{attribute 'linkalways'} 
{attribute 'no_explicit_call' := 'This FB is a CLASS and must be accessed using methods or properties'}
{attribute 'enable_dynamic_creation'}
FUNCTION_BLOCK BaseElement EXTENDS Disposable IMPLEMENTS I_EventEmitter, I_BaseElement
VAR
	inputPorts : InputPorts;
	outputPorts : OutputPorts;
	parameters : Parameters;
	contents : Contents;
	errors : Errors;
	extensions : Extensions;
	metadata : Metadata;
	eventEmitter : EventEmitter;
	disposables : Stack;
END_VAR

METHOD AddContent
VAR_INPUT
	Content : I_Content;
END_VAR
RegisterContent(Content);
END_METHOD

METHOD AddDataAsContent
VAR_INPUT
	Name : T_MAXSTRING;
	Data : I_Datatype;
END_VAR
VAR
	newContent : I_Content;
END_VAR
newContent := CreateContent(Name, Data);
RegisterDisposableToSelf(newContent);
END_METHOD

METHOD AddDataAsInputPort
VAR_INPUT
	Name : T_MAXSTRING;
	Data : I_Datatype;
END_VAR
VAR
	newInputPort : I_InputPort;
END_VAR
newInputPort := CreateInputPort(Name, Data);
RegisterDisposableToSelf(newInputPort);
END_METHOD

METHOD AddDataAsOutputPort
VAR_INPUT
	Name : T_MAXSTRING;
	Data : I_Datatype;
END_VAR
VAR
	newOutputPort : I_OutputPort;
END_VAR
newOutputPort := CreateOutputPort(Name, Data);
RegisterDisposableToSelf(newOutputPort);
END_METHOD

METHOD AddDataAsParameter
VAR_INPUT
	Name : T_MAXSTRING;
	Data : I_Datatype;
END_VAR
VAR
	newParameter : I_Parameter;
END_VAR
newParameter := CreateParameter(Name, Data);
RegisterDisposableToSelf(newParameter);
END_METHOD

METHOD AddError
VAR_INPUT
	Error : I_Error;
END_VAR
RegisterError(Error);
END_METHOD

METHOD AddExtension
VAR_INPUT
	Extension : I_Extension;
END_VAR
RegisterExtension(Extension);
END_METHOD

METHOD AddInputPort
VAR_INPUT
	InputPort : I_InputPort;
END_VAR
RegisterInputPort(InputPort);
END_METHOD

METHOD AddMetadatum
VAR_INPUT
	Metadatum : I_Metadatum;
END_VAR
RegisterMetadatum(Metadatum);
END_METHOD

METHOD AddOutputPort
VAR_INPUT
	OutputPort : I_OutputPort;
END_VAR
RegisterOutputPort(OutputPort);
END_METHOD

METHOD AddParameter
VAR_INPUT
	Parameter : I_Parameter;
END_VAR
RegisterParameter(Parameter);
END_METHOD

METHOD PROTECTED CreateContent : I_Content
VAR_INPUT
	ContentName : T_MAXSTRING;
	ContentData : I_Datatype;
END_VAR
VAR
	pContent : POINTER TO Content;
END_VAR
pContent := __NEW(Content(Name := ContentName, Data := ContentData, Parent := THIS^));
CreateContent := pContent^;
END_METHOD

METHOD PROTECTED CreateInputPort : I_InputPort
VAR_INPUT
	InputPortName : T_MAXSTRING;
	InputPortData : I_Datatype;
END_VAR
VAR
	pInputPort: POINTER TO InputPort;
END_VAR
pInputPort := __NEW(InputPort(Name := InputPortName, Data := InputPortData, Parent := THIS^));
CreateInputPort := pInputPort^;
END_METHOD

METHOD PROTECTED CreateOutputPort : I_OutputPort
VAR_INPUT
	OutputPortName : T_MAXSTRING;
	OutputPortData : I_Datatype;
END_VAR
VAR
	pOutputPort : POINTER TO OutputPort;
END_VAR
pOutputPort := __NEW(OutputPort(Name := OutputPortName, Data := OutputPortData, Parent := THIS^));
CreateOutputPort := pOutputPort^;
END_METHOD

METHOD PROTECTED CreateParameter : I_Parameter
VAR_INPUT
	ParameterName : T_MAXSTRING;
	ParameterData : I_Datatype;
END_VAR
VAR
	pParameter : POINTER TO Parameter;
END_VAR
pParameter := __NEW(Parameter(Name := ParameterName, Data := ParameterData, Parent := THIS^));
CreateParameter := pParameter^;
END_METHOD

METHOD PROTECTED DisposeAll : BOOL
VAR_INPUT
END_VAR
VAR
	disposable : I_Disposable;
END_VAR
WHILE disposables.TryPop(disposable) DO
	disposable.Dispose();
END_WHILE
END_METHOD

METHOD PROTECTED EmitOnContentAddedEvent
VAR_INPUT
	Content : I_Content;
END_VAR
VAR
	pContentAddedEvent : POINTER TO ContentAddedEvent;
END_VAR
IF Content = 0 THEN
	RETURN;
END_IF

pContentAddedEvent := __NEW(ContentAddedEvent(TargetContent := Content));
eventEmitter.Emit('OnContentAdded',pContentAddedEvent^);
pContentAddedEvent^.Dispose();
END_METHOD

METHOD PROTECTED EmitOnErrorAddedEvent
VAR_INPUT
	Error : I_Error;
END_VAR
VAR
	pErrorAddedEvent : POINTER TO ErrorAddedEvent;
END_VAR
IF Error = 0 THEN
	RETURN;
END_IF

pErrorAddedEvent := __NEW(ErrorAddedEvent(TargetError := Error));
eventEmitter.Emit('OnErrorAdded',pErrorAddedEvent^);
pErrorAddedEvent^.Dispose();
END_METHOD

METHOD PROTECTED EmitOnExtensionAddedEvent
VAR_INPUT
	Extension : I_Extension;
END_VAR
VAR
	pExtensionAddedEvent : POINTER TO ExtensionAddedEvent;
END_VAR
IF Extension = 0 THEN
	RETURN;
END_IF

pExtensionAddedEvent := __NEW(ExtensionAddedEvent(TargetExtension := Extension));
eventEmitter.Emit('OnExtensionAdded',pExtensionAddedEvent^);
pExtensionAddedEvent^.Dispose();
END_METHOD

METHOD PROTECTED EmitOnInputPortAddedEvent
VAR_INPUT
	InputPort : I_InputPort;
END_VAR
VAR
	pInputPortAddedEvent : POINTER TO InputPortAddedEvent;
END_VAR
IF InputPort = 0 THEN
	RETURN;
END_IF

pInputPortAddedEvent := __NEW(InputPortAddedEvent(TargetInputPort := InputPort));
eventEmitter.Emit('OnInputPortAdded',pInputPortAddedEvent^);
pInputPortAddedEvent^.Dispose();
END_METHOD

METHOD PROTECTED EmitOnMetadatumAddedEvent
VAR_INPUT
	Metadatum : I_Metadatum;
END_VAR
VAR
	pMetadatumAddedEvent : POINTER TO MetadatumAddedEvent;
END_VAR
IF Metadatum = 0 THEN
	RETURN;
END_IF

pMetadatumAddedEvent := __NEW(MetadatumAddedEvent(TargetMetadatum := Metadatum));
eventEmitter.Emit('OnMetadatumAdded',pMetadatumAddedEvent^);
pMetadatumAddedEvent^.Dispose();
END_METHOD

METHOD PROTECTED EmitOnOutputPortAddedEvent
VAR_INPUT
	OutputPort : I_OutputPort;
END_VAR
VAR
	pOutputPortAddedEvent : POINTER TO OutputPortAddedEvent;
END_VAR
IF OutputPort = 0 THEN
	RETURN;
END_IF

pOutputPortAddedEvent := __NEW(OutputPortAddedEvent(TargetOutputPort := OutputPort));
eventEmitter.Emit('OnOutputPortAdded',pOutputPortAddedEvent^);
pOutputPortAddedEvent^.Dispose();
END_METHOD

METHOD PROTECTED EmitOnParameterAddedEvent
VAR_INPUT
	Parameter : I_Parameter;
END_VAR
VAR
	pParameterAddedEvent : POINTER TO PropertyAddedEvent;
END_VAR
IF Parameter = 0 THEN
	RETURN;
END_IF

pParameterAddedEvent := __NEW(PropertyAddedEvent(TargetProperty := Parameter));
eventEmitter.Emit('OnParameterAdded',pParameterAddedEvent^);
pParameterAddedEvent^.Dispose();
END_METHOD

METHOD FB_exit : BOOL
VAR_INPUT
	bInCopyCode : BOOL; // if TRUE, the exit method is called for exiting an instance that is copied afterwards (online change).
END_VAR
IF bInCopyCode THEN
	RETURN;
END_IF

DisposeAll();
END_METHOD

METHOD PUBLIC GetContents : I_Contents
VAR_INPUT
END_VAR
GetContents := contents;
END_METHOD

METHOD PUBLIC GetErrors : I_Errors
VAR_INPUT
END_VAR
GetErrors := errors;
END_METHOD

METHOD PUBLIC GetExtensions : I_Extensions
VAR_INPUT
END_VAR
GetExtensions := extensions;
END_METHOD

METHOD PUBLIC GetInputPorts : I_InputPorts
VAR_INPUT
END_VAR
GetInputPorts := inputPorts;
END_METHOD

METHOD PUBLIC GetMetadata : I_Metadata
VAR_INPUT
END_VAR
GetMetadata := metadata;
END_METHOD

METHOD PUBLIC GetOutputPorts : I_OutputPorts
VAR_INPUT
END_VAR
GetOutputPorts := outputPorts;
END_METHOD

METHOD PUBLIC GetParameters : I_Parameters
VAR_INPUT
END_VAR
GetParameters := parameters;
END_METHOD

METHOD PUBLIC OffEvent
VAR_INPUT
	EventName : T_MaxString;
	EventHandler : I_EventHandler;
END_VAR
eventEmitter.OffEvent(EventName, EventHandler);
END_METHOD

METHOD PUBLIC OnceEvent
VAR_INPUT
	EventName : T_MaxString;
	EventHandler : I_EventHandler;
END_VAR
eventEmitter.OnceEvent(EventName, EventHandler);
END_METHOD

METHOD PUBLIC OnEvent
VAR_INPUT
	EventName : T_MaxString;
	EventHandler : I_EventHandler;
END_VAR
eventEmitter.OnEvent(EventName, EventHandler);
END_METHOD

METHOD PROTECTED RegisterContent
VAR_INPUT
	Content : I_Content;
END_VAR
contents.Insert(Content);
EmitOnContentAddedEvent(Content);
END_METHOD

METHOD PROTECTED RegisterDisposableToSelf
VAR_INPUT
	Disposable : I_Disposable;
END_VAR
disposables.Push(Disposable);
END_METHOD

METHOD PROTECTED RegisterError
VAR_INPUT
	Error : I_Error;
END_VAR
errors.Insert(Error);
EmitOnErrorAddedEvent(Error);
END_METHOD

METHOD PROTECTED RegisterExtension
VAR_INPUT
	Extension : I_Extension;
END_VAR
extensions.Insert(Extension);
EmitOnExtensionAddedEvent(Extension);
END_METHOD

METHOD PROTECTED RegisterInputPort
VAR_INPUT
	InputPort : I_InputPort;
END_VAR
inputPorts.Insert(InputPort);
EmitOnInputPortAddedEvent(InputPort);
END_METHOD

METHOD PROTECTED RegisterMetadatum
VAR_INPUT
	Metadatum : I_Metadatum;
END_VAR
metadata.Insert(Metadatum);
EmitOnMetadatumAddedEvent(Metadatum);
END_METHOD

METHOD PROTECTED RegisterOutputPort
VAR_INPUT
	OutputPort : I_OutputPort;
END_VAR
outputPorts.Insert(OutputPort);
EmitOnOutputPortAddedEvent(OutputPort);
END_METHOD

METHOD PROTECTED RegisterParameter
VAR_INPUT
	Parameter : I_Parameter;
END_VAR
parameters.Insert(Parameter);
EmitOnParameterAddedEvent(Parameter);
END_METHOD

METHOD PUBLIC SerializeWith
VAR_INPUT
	Serializer : I_Serializer;
END_VAR
Serializer.StartObject();
Serializer.AddKeyObject('inputPorts',inputPorts);
Serializer.AddKeyObject('outputPorts',outputPorts);
Serializer.AddKeyObject('parameters',parameters);
Serializer.AddKeyObject('contents',contents);
Serializer.AddKeyObject('errors',errors);
Serializer.AddKeyObject('extensions',extensions);
Serializer.AddKeyObject('metadata',metadata);
Serializer.EndObject();
END_METHOD

METHOD PROTECTED TryDeserializeExtensionsFrom : BOOL
VAR_INPUT
	Deserializer : I_Deserializer;
END_VAR
VAR
	extensionsDeserializer : I_Deserializer;
END_VAR
extensionsDeserializer := Deserializer.GetKey('extensions');
extensions.TryDeserializeFrom(extensionsDeserializer);
END_METHOD

METHOD PUBLIC TryDeserializeFrom : BOOL
VAR_INPUT
	Deserializer : I_Deserializer;
END_VAR
TryDeserializeFrom := 
	TryDeserializeParametersFrom(Deserializer) AND 
	TryDeserializeExtensionsFrom(Deserializer);
END_METHOD

METHOD PROTECTED TryDeserializeParametersFrom : BOOL
VAR_INPUT
	Deserializer : I_Deserializer;
END_VAR
VAR
	parametersDeserializer : I_Deserializer;
END_VAR
parametersDeserializer := Deserializer.GetKey('properties');
parameters.TryDeserializeFrom(parametersDeserializer);
END_METHOD

METHOD PUBLIC TryGetContentByName : BOOL
VAR_INPUT
	Name : T_MAXSTRING;
	Destination : REFERENCE TO I_Content;
END_VAR
VAR
	extensionName : T_MAXSTRING;
	extension : I_Extension;
	contentName : T_MAXSTRING;
END_VAR
IF Not HasExtensionNamespace(Name) THEN
	TryGetContentByName := contents.TryGetByName(Name,Destination);
	RETURN;
END_IF

extensionName := RemoveLastSegmentFromNamespace(Name);
contentName := GetLastSegmentFromNamespace(Name);

IF NOT TryGetExtensionByName(extensionName, extension) THEN
	RETURN;
END_IF

TryGetContentByName := extension.TryGetContentByName(contentName, Destination);
END_METHOD

METHOD PUBLIC TryGetExtensionByName : BOOL
VAR_INPUT
	Name : T_MAXSTRING;
	Destination : REFERENCE TO I_Extension;
END_VAR
VAR
	extensionName : T_MAXSTRING;
	remainingName : T_MAXSTRING;
	extension : I_Extension;
END_VAR
IF Not HasExtensionNamespace(Name) THEN
	TryGetExtensionByName := extensions.TryGetByName(Name, Destination);
	RETURN;
END_IF

extensionName := RemoveLastSegmentFromNamespace(Name);
remainingName := GetLastSegmentFromNamespace(Name);

IF NOT this^.TryGetExtensionByName(extensionName, extension) THEN
	RETURN;
END_IF

TryGetExtensionByName := extension.TryGetExtensionByName(remainingName, Destination);
END_METHOD

METHOD PUBLIC TryGetInputPortByName : BOOL
VAR_INPUT
	Name : T_MAXSTRING;
	Destination : REFERENCE TO I_InputPort;
END_VAR
VAR
	extensionName : T_MAXSTRING;
	extension : I_Extension;
	portName : T_MAXSTRING;
END_VAR
IF NOT HasExtensionNamespace(Name) THEN
	TryGetInputPortByName := inputPorts.TryGetByName(Name,Destination);
	RETURN;
END_IF

extensionName := RemoveLastSegmentFromNamespace(Name);
portName := GetLastSegmentFromNamespace(Name);

IF NOT TryGetExtensionByName(extensionName, extension) THEN
	RETURN;
END_IF

TryGetInputPortByName := extension.TryGetInputPortByName(portName, Destination);
END_METHOD

METHOD PUBLIC TryGetMetadatumByName : BOOL
VAR_INPUT
	Name : T_MAXSTRING;
	Destination : REFERENCE TO I_Metadatum;
END_VAR
VAR
	extensionName : T_MAXSTRING;
	extension : I_Extension;
	metadatumName : T_MAXSTRING;
END_VAR
IF NOT HasExtensionNamespace(Name) THEN
	TryGetMetadatumByName := metadata.TryGetByName(Name,Destination);
	RETURN;
END_IF

extensionName := RemoveLastSegmentFromNamespace(Name);
metadatumName := GetLastSegmentFromNamespace(Name);

IF NOT TryGetExtensionByName(extensionName, extension) THEN
	RETURN;
END_IF

TryGetMetadatumByName := extension.TryGetMetadatumByName(metadatumName, Destination);
END_METHOD

METHOD PUBLIC TryGetOutputPortByName : BOOL
VAR_INPUT
	Name : T_MAXSTRING;
	Destination : REFERENCE TO I_OutputPort;
END_VAR
VAR
	extensionName : T_MAXSTRING;
	extension : I_Extension;
	portName : T_MAXSTRING;
END_VAR
IF NOT HasExtensionNamespace(Name) THEN
	TryGetOutputPortByName := outputPorts.TryGetByName(Name,Destination);
	RETURN;
END_IF

extensionName := RemoveLastSegmentFromNamespace(Name);
portName := GetLastSegmentFromNamespace(Name);

IF NOT TryGetExtensionByName(extensionName, extension) THEN
	RETURN;
END_IF

TryGetOutputPortByName := extension.TryGetOutputPortByName(portName, Destination);
END_METHOD

METHOD PUBLIC TryGetParameterByName : BOOL
VAR_INPUT
	Name : T_MAXSTRING;
	Destination : REFERENCE TO I_Parameter;
END_VAR
VAR
	extensionName : T_MAXSTRING;
	extension : I_Extension;
	parameterName : T_MAXSTRING;
END_VAR
IF Not HasExtensionNamespace(Name) THEN
	TryGetParameterByName := parameters.TryGetByName(Name,Destination);
	RETURN;
END_IF

extensionName := RemoveLastSegmentFromNamespace(Name);
parameterName := GetLastSegmentFromNamespace(Name);

IF NOT TryGetExtensionByName(extensionName, extension) THEN
	RETURN;
END_IF

TryGetParameterByName := extension.TryGetParameterByName(parameterName, Destination);
END_METHOD

END_FUNCTION_BLOCK

(* stored: Version 1.1.0.1, ProductVersion 3.1.4024.12
   POU BaseElement: Id {65854565-5a7d-02f2-2709-1993949f09a2}, SpecialFunc None
   Folder Destructor: Id {8396773a-400b-43fa-8a6d-bbe9b1d6ecd3}
   Folder Protected: Id {48a95438-1d6b-0ead-29c1-c8ed21d5c5f8}
   Method AddContent: Id {65c5bac1-a3d0-002c-2cbe-a7b37fe3b45b}
   Method AddDataAsContent: Id {56e24acc-fc0e-4690-8a55-08bdbfb1feb3}
   Method AddDataAsInputPort: Id {4722f8e7-5165-4f79-9bed-1e281e05abb9}
   Method AddDataAsOutputPort: Id {dca4d70a-2386-4112-8b2e-e77a6edffbe6}
   Method AddDataAsParameter: Id {36004062-8b8a-4b3b-89b0-5b74d6f6bc9b}
   Method AddError: Id {4bbd3a02-551d-0fb6-097a-770c7ef9b02a}
   Method AddExtension: Id {12d5c379-9667-00ca-1a5e-59797e6bc21d}
   Method AddInputPort: Id {8aebf87c-0955-0d8e-0a5d-38af87c0ae0d}
   Method AddMetadatum: Id {371a7ce8-9ce1-0df1-08ad-592aac14c8db}
   Method AddOutputPort: Id {8d1e0294-027c-08af-0add-f26ea3b4e6b4}
   Method AddParameter: Id {22e10c77-042d-014a-1131-e8a94df32d37}
   Method CreateContent: Id {821b80ea-fa86-42dc-87c5-a687613888b2}
   Method CreateInputPort: Id {e170d3ea-2856-48fe-99f4-ab4fbe2d037c}
   Method CreateOutputPort: Id {bf3f2d9c-860a-4f77-a8dc-28e59fb38283}
   Method CreateParameter: Id {1ddc001e-24d0-48f3-b9e0-ff7f17397987}
   Method DisposeAll: Id {cb49ffb4-2cda-42c6-89fb-5c15e2905cfd}
   Method EmitOnContentAddedEvent: Id {982e38f9-d0ec-0d68-23b9-1014864696d7}
   Method EmitOnErrorAddedEvent: Id {5f18b0c5-cc95-02f2-100c-2ef3ad7e1a71}
   Method EmitOnExtensionAddedEvent: Id {f402631d-81f9-0a12-03bc-2a0bfe9edd1d}
   Method EmitOnInputPortAddedEvent: Id {999a27ba-e180-0c81-3fd5-7f26e1dcafa9}
   Method EmitOnMetadatumAddedEvent: Id {5e041b08-cbe4-0f2d-0996-099d35827b7a}
   Method EmitOnOutputPortAddedEvent: Id {0092de63-0b62-04d1-3582-5fcf00057f98}
   Method EmitOnParameterAddedEvent: Id {ef9a119a-00ba-01e3-3336-a5211fd3bf30}
   Method FB_exit: Id {6b932cb7-4150-4273-8597-9e500c0eaf5e}
   Method GetContents: Id {81f125c5-c13a-026a-3de6-aa1ebc6668c9}
   Method GetErrors: Id {0627fae9-4882-0c55-17d9-c59657d05963}
   Method GetExtensions: Id {be4c5a1a-53d3-0499-27b1-32409495df61}
   Method GetInputPorts: Id {7de9fbdd-fa4d-0d6e-0b3b-13feae4c89d5}
   Method GetMetadata: Id {dbde985b-051a-0727-258a-c2925ede1d19}
   Method GetOutputPorts: Id {f627e22a-94e0-005f-10c4-a9f76f86d6e8}
   Method GetParameters: Id {f803076c-9d09-002d-18bd-949f984e4d58}
   Method OffEvent: Id {3826f2c5-8817-085f-32d4-f42ca6017d84}
   Method OnceEvent: Id {c0653d6f-a473-06ad-0f4f-23e16a4ab170}
   Method OnEvent: Id {f1641710-5271-0c90-204a-d8ba0111dbe4}
   Method RegisterContent: Id {b67f9558-618d-4bfd-b717-886a90f2936b}
   Method RegisterDisposableToSelf: Id {818ccf26-b9c1-40b3-8452-6ca75c4281c5}
   Method RegisterError: Id {65cdee1a-3625-45b6-bfd7-f72ce4f3aef5}
   Method RegisterExtension: Id {f527d3d7-1297-4450-90c8-dbf3475e7a3d}
   Method RegisterInputPort: Id {a90f95fc-e99b-45fe-ad6f-5621929e0e45}
   Method RegisterMetadatum: Id {c3fb64d8-e827-436e-9972-728da0497a0c}
   Method RegisterOutputPort: Id {8be6e625-9fd4-44dd-a437-f152d0338e1b}
   Method RegisterParameter: Id {8ed8ffd2-775b-4ca8-bf44-de6ba556c507}
   Method SerializeWith: Id {41b86bad-3ef8-4c80-9f08-2299a4ef627c}
   Method TryDeserializeExtensionsFrom: Id {ad9e3ab9-6d42-4e27-a29c-b45a0249832c}
   Method TryDeserializeFrom: Id {520fe007-9bcd-4e66-88a2-2aa342fc675e}
   Method TryDeserializeParametersFrom: Id {c54ae027-05a9-42d5-aace-677f13db3ada}
   Method TryGetContentByName: Id {5ed45c1e-e709-063a-078b-c4ffa6e05f7e}
   Method TryGetExtensionByName: Id {40285acc-4e71-0188-0b28-516f73de9f1d}
   Method TryGetInputPortByName: Id {f48a519d-be51-089e-1869-f8f4fa949214}
   Method TryGetMetadatumByName: Id {a3a91194-7db2-0843-24e0-73a63eb18407}
   Method TryGetOutputPortByName: Id {e92ddf93-b96a-08ad-01fb-739fc2280c59}
   Method TryGetParameterByName: Id {f428aa13-e6f6-0562-2045-054d9aa11372} *)
